(* IEC 61131-3 sources: POMIRTS_lab3/AS/Library/AsCisMan, 3 files *)

(* ---- AsCisMan.typ ---- *)
(********************************************************************
 * COPYRIGHT -- Bernecker + Rainer
 ********************************************************************
 * Library: AsCisMan
 * File: AsCisMan.typ
 * Author: B+R
 ********************************************************************
 * Data types of library AsCisMan
 ********************************************************************)

TYPE
	vfAxisInfo_typ : STRUCT								(*statistics and internal information*)
		Device	: STRING[20] ;							(*interface device string*)
		Mode	: STRING[20] ;							(*interface mode string*)
		Typ	: UINT ;									(*device type*)
		IndexVf	: USINT ;								(*internal array index for axis structure*)
		IndexIf	: USINT ;								(*internal array index for interface structure*)
		VersionLib	: ARRAY[0..9] OF USINT ;			(*version of the AsCisMan.br library*)
		VersionDrv	: ARRAY[0..9] OF USINT ;			(*version of the driver task cis_vf.br or cis_ps.br*)
		VersionOsVf	: ARRAY[0..9] OF USINT ;			(*version of the cis_osvf operating system transferred to the VF*)
		VersionData	: ARRAY[0..9] OF USINT ;			(*data object version*)
		VfPNominal	: UINT ;							(*nominal power of the VF module in W (read from the VF EPROM)*)
		VfModuleID	: UINT ;							(*ID number of the VF module (read from the VF EPROM)*)
		VfSerialNr	: UDINT ;							(*serial number of the VF module (read from the VF EPROM)*)
		VfCurrentLSB	: UINT ;						(*current resolution of VF module in mA/Bit (read from the VF EPROM)*)
		CyclesPowerOn	: UINT ;						(*counter for the number of power ons*)
		HoursPowerOn	: UDINT ;						(*counter for the hours that voltage is applied to the VF module*)
		HoursMotorOn	: UDINT ;						(*counter for the hours the motor has power*)
		MinutesPowerOn	: USINT ;						(*counter minutes of VF module under voltage (incremented to 254 only once)*)
		MinutesMotorOn	: USINT ;						(*counter minutes of powered motor (incremented to 254 only once)*)
		HistoryMaxTempIGBT	: USINT ;					(*overall maximum IGBT temperature in degree celsius*)
		HistoryMaxTempMotor	: USINT ;					(*overall maximum motor temperature in degree celsius*)
		HistoryMaxTempCPU1	: USINT ;					(*overall maximum CPU temperature1 in degree celsius*)
		HistoryMaxTempCPU2	: USINT ;					(*overall maximum CPU temperature2 in degree celsius*)
		HistoryMaxCurrent	: UINT ;					(*overall maximum DC bus current in mA*)
		HistoryMaxUDCLink	: UINT ;					(*overall maximum DC bus voltage in VCD*)
		HistoryChangedSlot	: USINT ;					(*counter VF module inserted in different slot than at the last power on*)
		HistoryChangedPS	: USINT ;					(*counter VF module inserted in different CIS PS than at the last power on*)
		FactUDCLink	: REAL ;							(*DC bus voltage measurement correction factor (0.880-1.120)*)
		IdentXOpen	: UDINT ;							(*internal use*)
		StatusXOpen	: UINT ;							(*internal use*)
		IdentData	: UDINT ;							(*internal use*)
		pData	: UDINT ;								(*internal use*)
		lenData	: UDINT ;								(*internal use*)
		StatusData	: UINT ;							(*internal use*)
	END_STRUCT;
	vfAxisNetwork_typ : STRUCT							(*network and individual parameter operations*)
		Init	: USINT ;								(*initializes the connection (FU responds to the driver)*)
		ParIDRequest	: USINT ;						(*sets/reads FI parameters: requested ID*)
		ParIDResponse	: USINT ;						(*sets/reads individual parameters: response from read/write ID*)
		ParData	: UINT ;								(*sets/reads individual parameters depending on the parameter: data*)
		EPromAdrRequest	: USINT ;						(*sets/reads byte at EEPROM: requested address ($00…$7F reserved for OS)*)
		EPromAdrResponse	: USINT ;					(*sets/reads EEPROM bytes: response from read/write address*)
		EPromData	: USINT ;							(*sets/reads EEPROM : Data*)
	END_STRUCT;
	vfAxisParaVf_typ : STRUCT							(*parameter*)
		UDCNominal	: UINT ;							(*nominal DC bus voltage*)
		VfCurveV	: ARRAY[0..7] OF UINT ;				(*v/f curve array (voltage point 0-7)*)
		VfCurveF	: ARRAY[0..7] OF UINT ;				(*v/f curve array (frequency point 0-7)*)
		FreqMax	: UINT ;								(*maximum frequency*)
		MaxCurrent	: UINT ;							(*DC bus current limit*)
		IntAccRamp	: UINT ;							(*internal acceleration ramp (corresponds to about 5 ms/step)*)
		IntDecRamp	: UINT ;							(*internal deceleration ramp (corresponds to about 5 ms/step)*)
		TimeStopped	: UINT ;							(*time between the motor's stopping and status, stopped = 1*)
		ModeStopped	: USINT ;							(*ModeStopped=0..speed takes effect immediately, ModeStopped=1..speed takes effect only when status*)
		Pwm	: USINT ;									(*frequency for pulse width modulation (currently fixed at 5 kHz)*)
		TorqueCtrl	: USINT ;							(*enable VF torque check*)
		TempMotorMax	: USINT ;						(*maximum motor temperature*)
		CurErrorAutoAck	: USINT ;						(*enables automatic acknowledgement of overcurrent errors*)
		spare1	: USINT ;								(*free*)
		UDCMax	: UINT ;								(*maximum permissible DC bus voltage: 0...default value 760VDC is used*)
	END_STRUCT;
	vfAxisParaTemp_typ : STRUCT							(*parameter*)
		R0	: UINT ;									(*resistance for T[0]*)
		R7	: UINT ;									(*resistance for T[7]*)
		T	: ARRAY[0..7] OF SINT ;						(*field for temperature*)
	END_STRUCT;
	vfAxisPara_typ : STRUCT								(*parameter*)
		Vf	: vfAxisParaVf_typ ;						(*CIS FU parameters*)
		Temp	: vfAxisParaTemp_typ ;					(*motor temperature sensor parameter*)
	END_STRUCT;
	vfAxisMove_typ : STRUCT								(*motion*)
		Speed	: DINT ;								(*target speed [0.01Hz] (-600.00…600.00Hz)*)
		CurrLimit	: UINT ;							(*DC bus current limit (0…65000mA)*)
		UDCInject	: UINT ;							(*DC brake voltage (for StopMode=2 only)*)
		StopMode	: USINT ;							(*is given es a target speed, e.g. 0...motor loses current immediately and spins out*)
		AccPos	: UDINT ;								(*acceleration in a positive direction [0.01Hz/s] (0.01…1000.00Hz/s)*)
		AccNeg	: UDINT ;								(*acceleration in a negative direction [0.01Hz/s] (0.01…1000.00Hz/s)*)
		DecPos	: UDINT ;								(*deceleration in a positive direction [0.01Hz/s] (0.01…1000.00Hz/s)*)
		DecNeg	: UDINT ;								(*deceleration in a negative direction [0.01Hz/s] (0.01…1000.00Hz/s)*)
	END_STRUCT;
	vfAxisStatus_typ : STRUCT							(*status*)
		SpeedRamped	: DINT ;							(*current ramp speed being sent to the FC (unit = 0.01Hz)*)
		UDCInject	: UINT ;							(*currently induced braking voltage in V*)
		ActTempIGBT	: USINT ;							(*current FC-IGBT temperature in degree celsius*)
		MaxTempIGBT	: USINT ;							(*maximum FC-IGBT temperature in degree celsius*)
		ActTempMotor	: USINT ;						(*current FC motor temperature in degree celsius*)
		MaxTempMotor	: USINT ;						(*maximum FC motor temperature in degree celsius*)
		ActTempRect	: USINT ;							(*current bridge rectifier temperature in degree celsius*)
		MaxTempRect	: USINT ;							(*maximum bridge rectifier temperature in degree celsius*)
		ActTempPS	: USINT ;							(*current internal temperature in degree celsius*)
		MaxTempPS	: USINT ;							(*maximum internal temperature in degree celsius*)
		ActTempCPU1	: USINT ;							(*current internal CIS CPU temperature 1 in degree celsius (up to 80degree OK)*)
		MaxTempCPU1	: USINT ;							(*maximum internal CIS CPU temperature 1 in degree celsius*)
		ActTempCPU2	: USINT ;							(*current internal CIS CPU temperature 2 in degree celsius (up to 80degree OK)*)
		MaxTempCPU2	: USINT ;							(*maximum internal CIS CPU temperature 2 in degree celsius*)
		ActCurrent	: UINT ;							(*current IGBT DC bus current in mA*)
		MaxCurrent	: UINT ;							(*maximum IGBT DC bus current in mA*)
		ActUDCLink	: UINT ;							(*current FC DC bus voltage in VDC*)
		MaxUDCLink	: UINT ;							(*maximum FC DC bus voltage in VDC*)
		CPU	: UINT ;									(*statusBits CPU*)
		CISPS1	: USINT ;								(*statusBits1 FC basis board*)
		CISPS2	: USINT ;								(*statusBits2 FC basis board*)
		Stopped	: USINT ;								(*Motor stopped (current rotor speed = 0 detected)*)
		Active	: USINT ;								(*FC active (cyclic speed assignment to CIS FC is active)*)
		ParaInit	: USINT ;							(*Parameter initialized*)
		PowerOk	: USINT ;								(*DC bus voltage OK*)
	END_STRUCT;
	vfAxisError_typ : STRUCT							(*error*)
		Active	: USINT ;								(*cumulative error: at least one error is active*)
		Current	: USINT ;								(*DC bus current over current limit (warning)*)
		CurrentOff	: USINT ;							(*DC bus current too high - FC stopped, error must be acknowledged*)
		TempIGBT	: USINT ;							(*IGBT temperature warning*)
		TempIGBTOff	: USINT ;							(*IGBT temperature too high - FC stopped, error must be acknowledged*)
		TempMotor	: USINT ;							(*motor temperature warning*)
		TempMotorOff	: USINT ;						(*motor temperature too high - FC stopped, error must be acknowledged*)
		TempMotorBreak	: USINT ;						(*motor temperature sensor wire break*)
		TempMotorShort	: USINT ;						(*motor temperature sensor short circuit*)
		VoltageHigh	: USINT ;							(*DC bus voltage too high*)
		Amplifier	: USINT ;							(*IGBT control internal error*)
		cntComTimeOff	: UDINT ;						(*counter: milliseconds that have passed since the last valid response from the FC*)
		cntCom	: UINT ;								(*counter communication error: communication timeout*)
		cntCommand	: UINT ;							(*counter communication error: illegal command*)
		cntParameter	: UINT ;						(*counter communication error: parameter outside of the permitted range*)
		cntService	: UINT ;							(*counter communication error: illegal service command*)
		cntAcknowledge	: UINT ;						(*counter communication error: could not acknowledge error - error still active*)
		cntCheckSumVFD	: UINT ;						(*counter checksum error (illegal checksum in FC data)*)
		cntEpromLock	: UINT ;						(*counter communication error: EPROM access blocked*)
		cntAmplitudeDelta	: UINT ;					(*counter error in VF curve parameters (voltage amplitude not climbing monotonously)*)
		cntFrequencyDelta	: UINT ;					(*counter error in VF curve parameters (frequency not climbing monotonously)*)
		cntLifeSignal	: UINT ;						(*counter: FC didn't receive any valid data for 200 ms*)
		cntCheckSumCPU	: UINT ;						(*counter checksum error (illegal checksum in FC data)*)
		cntResponsePara	: UINT ;						(*counter communication error (illegal data in response telegram)*)
		cntResponseSpd	: UINT ;						(*counter communication error (illegal data in response telegram)*)
		cntResponseError	: UINT ;					(*counter communication error (illegal data in response telegram)*)
	END_STRUCT;
	vfAxisInterntOut_typ : STRUCT						(*internal use*)
		IN	: BOOL ;
		PT	: UDINT ;
		Q	: BOOL ;
		ET	: UDINT ;
		StartTime	: UDINT ;
		M	: BOOL ;
	END_STRUCT;
	vfAxisInternal_typ : STRUCT							(*internal use*)
		cmdSubject	: UINT ;							(*handshake for the vfaction() function: command subject*)
		cmdAction	: UINT ;							(*handshake for the vfaction() function: command action*)
		cmdPara	: USINT ;								(*handshake for the vfaction() function: command related parameterID*)
		cmdData	: UINT ;								(*handshake for the vfaction() function: command related data*)
		cntStep	: USINT ;								(*internal step*)
		Write	: USINT ;								(*0..process command, 1..send frame, 2..wait for response*)
		BufWrite	: ARRAY[0..5] OF USINT ;			(*buffer for the sent frame*)
		BufRead	: ARRAY[0..5] OF USINT ;				(*buffer for the received frame*)
		Sequence	: USINT ;							(*indicates the class of parameter ID*)
		cntInitEpromRead	: USINT ;					(*counter for read EPROM data during initialization*)
		cntInitUfCurveSet	: USINT ;					(*counter for sent U/f data*)
		tOut	: vfAxisInterntOut_typ ;				(*receive timeout*)
		ActTempMotorR	: UINT ;						(*measured resistance of the motor temperature sensor*)
		MaxTempMotorR	: UINT ;						(*measured resistance of the motor temperature sensor*)
		TempMotorRFilter	: ARRAY[0..9] OF UINT ;		(*filter buffer for motor temperature filters*)
		cntTempMotorRFilter	: UINT ;					(*filter counter for motor temperature filters*)
		OldUDCInject	: UINT ;						(*UDCInject edge*)
		SpeedRamped	: REAL ;							(*output of the speed ramp in REAL*)
		TestFan	: USINT ;								(*=1 for manually testing the internal fans*)
		cntInfoWrite	: USINT ;						(*counter*)
		CyclesPowerOnCheck	: UINT ;					(*EPROM: backup copy of Info.CyclesPowerOn*)
		HoursPowerOnCheck	: UDINT ;					(*EPROM: backup copy of Info.HoursPowerOn*)
		HoursMotorOnCheck	: UDINT ;					(*EPROM: backup copy of Info.HoursMotorOn*)
		HistoryBufferAdr	: ARRAY[0..15] OF USINT ;	(*history address storage*)
		HistoryBufferData	: ARRAY[0..15] OF USINT ;	(*history data storage*)
		HistoryBufferCnt	: USINT ;					(*counter for pending historical data*)
		HistorySlot	: USINT ;							(*EPROM: VF inserted in slot number*)
		HistoryMacId	: ARRAY[0..2] OF USINT ;		(*EPROM: MacID of the CIS-PS*)
		HistoryMacIdChecksum	: USINT ;				(*EPROM: MacID checksum*)
		FactUDCLink	: REAL ;							(*EPROM: DC bus voltage measurement correction factor*)
	END_STRUCT;
	vfAXIS_typ : STRUCT									(*AXIS information*)
		Info	: vfAxisInfo_typ ;						(*statistics and internal information*)
		Network	: vfAxisNetwork_typ ;					(*network and individual parameter operations*)
		Para	: vfAxisPara_typ ;						(*parameter*)
		Move	: vfAxisMove_typ ;						(*motion*)
		Status	: vfAxisStatus_typ ;					(*status*)
		Error	: vfAxisError_typ ;						(*error*)
		Internal	: vfAxisInternal_typ ;				(*internal use*)
	END_STRUCT;
	vfInterfaceBuf_typ : STRUCT							(*internal use*)
		Byte0	: USINT ;
		Command	: USINT ;
		ByteHI	: USINT ;
		ByteLO	: USINT ;
		CheckSum	: USINT ;
		spare0	: USINT ;
	END_STRUCT;
	vfInterface_typ : STRUCT							(*internal use*)
		Ident	: UDINT ;
		cntFrame	: USINT ;
		oldFrame	: USINT ;
		cntBufWrite	: USINT ;
		cntBufRead	: USINT ;
		cntFrameWrite	: USINT ;
		cntFrameRead	: USINT ;
		FrameRead	: ARRAY[0..7] OF USINT ;
		cntFrameRead85	: USINT ;
		FrameRead85	: ARRAY[0..1] OF USINT ;
		BufWrite	: ARRAY[0..7] OF vfInterfaceBuf_typ ;
		BufRead	: ARRAY[0..7] OF vfInterfaceBuf_typ ;
	END_STRUCT;
	vfDebug_typ : STRUCT								(*internal use*)
		Time	: UDINT ;
		UDC	: UINT ;
		Current	: UINT ;
		Temp	: USINT ;
		BufferSend	: ARRAY[0..4] OF USINT ;
		BufferRecv	: ARRAY[0..11] OF USINT ;
		BufferRecvNb	: USINT ;
		ErrorCom	: USINT ;
		ErrorCheckFU	: USINT ;
		ErrorCheckCPU	: USINT ;
		ErrorCommand	: USINT ;
		ErrorParameter	: USINT ;
		ErrorService	: USINT ;
		ErrorResponse	: USINT ;
		ErrorAcknowledge	: USINT ;
		ErrorEpromLock	: USINT ;
		ErrorAmplitudeDelta	: USINT ;
		ErrorFrequencyDelta	: USINT ;
		ErrorLifeSignal	: USINT ;
	END_STRUCT;
	vfDebugResponse_typ : STRUCT						(*internal use*)
		Write	: ARRAY[0..5] OF USINT ;
		Read	: ARRAY[0..5] OF USINT ;
	END_STRUCT;
	vfErrorTrace_typ : STRUCT							(*internal use*)
		Fu	: USINT ;
		Error	: USINT ;
		Time	: UDINT ;
	END_STRUCT;
END_TYPE

(* ---- AsCisMan.fun ---- *)
(********************************************************************
 * COPYRIGHT -- Bernecker + Rainer
 ********************************************************************
 * Library: AsCisMan
 * File: AsCisMan.fun
 * Author: B+R
 ********************************************************************
 * Functions and function blocks of library AsCisMan
 ********************************************************************)

FUNCTION_BLOCK initps05								(*boots and allocates a CIS base unit 80CIS.PS0-5 (7 slot, 6.5 kW)*)
	VAR_INPUT
		Enable	:BOOL;								(*enables execution*)
		ParaVF1	:STRING[8];							(*name of the slot1 initialization parameter data object*)
		ParaVF2	:STRING[8];							(*name of the slot2 initialization parameter data object*)
		ParaVF3	:STRING[8];							(*name of the slot3 initialization parameter data object*)
		ParaVF4	:STRING[8];							(*name of the slot4 initialization parameter data object*)
		ParaVF5	:STRING[8];							(*name of the slot5 initialization parameter data object*)
		ParaVF6	:STRING[8];							(*name of the slot6 initialization parameter data object*)
		ParaVF7	:STRING[8];							(*name of the slot7 initialization parameter data object*)
	END_VAR
	VAR_OUTPUT
		Status	:UINT;								(*execution status: ERR_OK, ERR_FUB_ENABLE_FALSE, 0xXXXX = see help*)
		IdentCPU	:UDINT;							(*identifier for the CPU data (for use with run_cpu)*)
		IdentVF1	:UDINT;							(*identifier for the VF slot 1 (for use with run_vfx)*)
		IdentVF2	:UDINT;							(*identifier for the VF slot 2 (for use with run_vfx)*)
		IdentVF3	:UDINT;							(*identifier for the VF slot 3 (for use with run_vfx)*)
		IdentVF4	:UDINT;							(*identifier for the VF slot 4 (for use with run_vfx)*)
		IdentVF5	:UDINT;							(*identifier for the VF slot 5 (for use with run_vfx)*)
		IdentVF6	:UDINT;							(*identifier for the VF slot 6 (for use with run_vfx)*)
		IdentVF7	:UDINT;							(*identifier for the VF slot 7 (for use with run_vfx)*)
		BootOkBitsVF	:USINT;						(*bit-coded status: bit=0...boot failed, bit=1...boot successful*)
	END_VAR
	VAR
		Object	:ARRAY[0..8] OF UDINT;				(*internal variable*)
		StatusAlloc	:ARRAY[0..8] OF UINT;			(*internal variable*)
			vf_bsl_00	:vf_bsl;					(*internal variable*)
			vf_bsl_01	:vf_bsl;					(*internal variable*)
		vf_bsl_02	:vf_bsl;						(*internal variable*)
		vf_bsl_03	:vf_bsl;						(*internal variable*)
		vf_bsl_04	:vf_bsl;						(*internal variable*)
		vf_bsl_05	:vf_bsl;						(*internal variable*)
		vf_bsl_06	:vf_bsl;						(*internal variable*)
		vf_bsl_07	:vf_bsl;						(*internal variable*)
		vf_bsl_08	:vf_bsl;						(*internal variable*)
		zzvfalloc00000	:vfalloc;					(*internal variable*)
		zzvfalloc00001	:vfalloc;					(*internal variable*)
		zzvfalloc00002	:vfalloc;					(*internal variable*)
		zzvfalloc00003	:vfalloc;					(*internal variable*)
		zzvfalloc00004	:vfalloc;					(*internal variable*)
		zzvfalloc00005	:vfalloc;					(*internal variable*)
		zzvfalloc00006	:vfalloc;					(*internal variable*)
		zzvfalloc00007	:vfalloc;					(*internal variable*)
	END_VAR
END_FUNCTION_BLOCK

FUNCTION_BLOCK initps04								(*boots and allocates a CIS base unit 80CIS.PS0-4 (4 slot, 16 kW)*)
	VAR_INPUT
		Enable	:BOOL;								(*enables execution*)
		ParaVF1	:STRING[8];							(*name of the slot1 initialization parameter data object*)
		ParaVF2	:STRING[8];							(*name of the slot2 initialization parameter data object*)
		ParaVF3	:STRING[8];							(*name of the slot3 initialization parameter data object*)
		ParaVF4	:STRING[8];							(*name of the slot4 initialization parameter data object*)
	END_VAR
	VAR_OUTPUT
		Status	:UINT;								(*execution status: ERR_OK, ERR_FUB_ENABLE_FALSE, 0xXXXX = see help*)
		IdentCPU	:UDINT;							(*identifier for the CPU data (for use with run_cpu)*)
		IdentVF1	:UDINT;							(*identifier for the VF slot 1 (for use with run_vfx)*)
		IdentVF2	:UDINT;							(*identifier for the VF slot 2 (for use with run_vfx)*)
		IdentVF3	:UDINT;							(*identifier for the VF slot 3 (for use with run_vfx)*)
		IdentVF4	:UDINT;							(*identifier for the VF slot 4 (for use with run_vfx)*)
		BootOkBitsVF	:USINT;						(*bit-coded status: bit=0...boot failed, bit=1...boot successful*)
	END_VAR
	VAR
		Object	:ARRAY[0..8] OF UDINT;				(*internal variable*)
		StatusAlloc	:ARRAY[0..8] OF UINT;			(*internal variable*)
		vf_bsl_00	:vf_bsl;						(*internal variable*)
		vf_bsl_01	:vf_bsl;						(*internal variable*)
		vf_bsl_02	:vf_bsl;						(*internal variable*)
		vf_bsl_03	:vf_bsl;						(*internal variable*)
		vf_bsl_08	:vf_bsl;						(*internal variable*)
		zzvfalloc00000	:vfalloc;					(*internal variable*)
		zzvfalloc00001	:vfalloc;					(*internal variable*)
		zzvfalloc00002	:vfalloc;					(*internal variable*)
		zzvfalloc00003	:vfalloc;					(*internal variable*)
		zzvfalloc00004	:vfalloc;					(*internal variable*)
	END_VAR
END_FUNCTION_BLOCK

FUNCTION_BLOCK initps03								(*boots and allocates a CIS base unit 80CIS.PS0-3 (8 slot, 16 kW)*)
	VAR_INPUT
		Enable	:BOOL;								(*enables execution*)
		ParaVF1	:STRING[8];							(*name of the slot1 initialization parameter data object*)
		ParaVF2	:STRING[8];							(*name of the slot2 initialization parameter data object*)
		ParaVF3	:STRING[8];							(*name of the slot3 initialization parameter data object*)
		ParaVF4	:STRING[8];							(*name of the slot4 initialization parameter data object*)
		ParaVF5	:STRING[8];							(*name of the slot5 initialization parameter data object*)
		ParaVF6	:STRING[8];							(*name of the slot6 initialization parameter data object*)
		ParaVF7	:STRING[8];							(*name of the slot7 initialization parameter data object*)
		ParaVF8	:STRING[8];							(*name of the slot8 initialization parameter data object*)
	END_VAR
	VAR_OUTPUT
		Status	:UINT;								(*execution status: ERR_OK, ERR_FUB_ENABLE_FALSE, 0xXXXX = see help*)
		IdentCPU	:UDINT;							(*identifier for the CPU data (for use with run_cpu)*)
		IdentVF1	:UDINT;							(*identifier for the VF slot 1 (for use with run_vfx)*)
		IdentVF2	:UDINT;							(*identifier for the VF slot 2 (for use with run_vfx)*)
		IdentVF3	:UDINT;							(*identifier for the VF slot 3 (for use with run_vfx)*)
		IdentVF4	:UDINT;							(*identifier for the VF slot 4 (for use with run_vfx)*)
		IdentVF5	:UDINT;							(*identifier for the VF slot 5 (for use with run_vfx)*)
		IdentVF6	:UDINT;							(*identifier for the VF slot 6 (for use with run_vfx)*)
		IdentVF7	:UDINT;							(*identifier for the VF slot 7 (for use with run_vfx)*)
		IdentVF8	:UDINT;							(*identifier for the VF slot 8 (for use with run_vfx)*)
		BootOkBitsVF	:USINT;						(*bit-coded status: bit=0...boot failed, bit=1...boot successful*)
	END_VAR
	VAR
		Object	:ARRAY[0..8] OF UDINT;				(*internal variable*)
		StatusAlloc	:ARRAY[0..8] OF UINT;			(*internal variable*)
		vf_bsl_00	:vf_bsl;						(*internal variable*)
		vf_bsl_01	:vf_bsl;						(*internal variable*)
		vf_bsl_02	:vf_bsl;						(*internal variable*)
		vf_bsl_03	:vf_bsl;						(*internal variable*)
		vf_bsl_04	:vf_bsl;						(*internal variable*)
		vf_bsl_05	:vf_bsl;						(*internal variable*)
		vf_bsl_06	:vf_bsl;						(*internal variable*)
		vf_bsl_07	:vf_bsl;						(*internal variable*)
		vf_bsl_08	:vf_bsl;						(*internal variable*)
		zzvfalloc00000	:vfalloc;					(*internal variable*)
		zzvfalloc00001	:vfalloc;					(*internal variable*)
		zzvfalloc00002	:vfalloc;					(*internal variable*)
		zzvfalloc00003	:vfalloc;					(*internal variable*)
		zzvfalloc00004	:vfalloc;					(*internal variable*)
		zzvfalloc00005	:vfalloc;					(*internal variable*)
		zzvfalloc00006	:vfalloc;					(*internal variable*)
		zzvfalloc00007	:vfalloc;					(*internal variable*)
		zzvfalloc00008	:vfalloc;					(*internal variable*)
	END_VAR
END_FUNCTION_BLOCK

FUNCTION_BLOCK initps02								(*boots and allocates a CIS base unit 80CIS.PS0-2 (8 slot, 8 kW)*)
	VAR_INPUT
		Enable	:BOOL;								(*enables execution*)
		ParaVF1	:STRING[8];							(*name of the slot1 initialization parameter data object*)
		ParaVF2	:STRING[8];							(*name of the slot2 initialization parameter data object*)
		ParaVF3	:STRING[8];							(*name of the slot3 initialization parameter data object*)
		ParaVF4	:STRING[8];							(*name of the slot4 initialization parameter data object*)
		ParaVF5	:STRING[8];							(*name of the slot5 initialization parameter data object*)
		ParaVF6	:STRING[8];							(*name of the slot6 initialization parameter data object*)
		ParaVF7	:STRING[8];							(*name of the slot7 initialization parameter data object*)
		ParaVF8	:STRING[8];							(*name of the slot8 initialization parameter data object*)
	END_VAR
	VAR_OUTPUT
		Status	:UINT;								(*execution status: ERR_OK, ERR_FUB_ENABLE_FALSE, 0xXXXX = see help*)
		IdentCPU	:UDINT;							(*identifier for the CPU data (for use with run_cpu)*)
		IdentVF1	:UDINT;							(*identifier for the VF slot 1 (for use with run_vfx)*)
		IdentVF2	:UDINT;							(*identifier for the VF slot 2 (for use with run_vfx)*)
		IdentVF3	:UDINT;							(*identifier for the VF slot 3 (for use with run_vfx)*)
		IdentVF4	:UDINT;							(*identifier for the VF slot 4 (for use with run_vfx)*)
		IdentVF5	:UDINT;							(*identifier for the VF slot 5 (for use with run_vfx)*)
		IdentVF6	:UDINT;							(*identifier for the VF slot 6 (for use with run_vfx)*)
		IdentVF7	:UDINT;							(*identifier for the VF slot 7 (for use with run_vfx)*)
		IdentVF8	:UDINT;							(*identifier for the VF slot 8 (for use with run_vfx)*)
		BootOkBitsVF	:USINT;						(*bit-coded status: bit=0...boot failed, bit=1...boot successful*)
	END_VAR
	VAR
		Object	:ARRAY[0..8] OF UDINT;				(*internal variable*)
		StatusAlloc	:ARRAY[0..8] OF UINT;			(*internal variable*)
		vf_bsl_00	:vf_bsl;						(*internal variable*)
		vf_bsl_01	:vf_bsl;						(*internal variable*)
		vf_bsl_02	:vf_bsl;						(*internal variable*)
		vf_bsl_03	:vf_bsl;						(*internal variable*)
		vf_bsl_04	:vf_bsl;						(*internal variable*)
		vf_bsl_05	:vf_bsl;						(*internal variable*)
		vf_bsl_06	:vf_bsl;						(*internal variable*)
		vf_bsl_07	:vf_bsl;						(*internal variable*)
		vf_bsl_08	:vf_bsl;						(*internal variable*)
		zzvfalloc00000	:vfalloc;					(*internal variable*)
		zzvfalloc00001	:vfalloc;					(*internal variable*)
		zzvfalloc00002	:vfalloc;					(*internal variable*)
		zzvfalloc00003	:vfalloc;					(*internal variable*)
		zzvfalloc00004	:vfalloc;					(*internal variable*)
		zzvfalloc00005	:vfalloc;					(*internal variable*)
		zzvfalloc00006	:vfalloc;					(*internal variable*)
		zzvfalloc00007	:vfalloc;					(*internal variable*)
		zzvfalloc00008	:vfalloc;					(*internal variable*)
	END_VAR
END_FUNCTION_BLOCK

FUNCTION_BLOCK run_cpu								(*communicates cyclic to the CPU*)
	VAR_INPUT
		Enable	:BOOL;								(*enables execution*)
		IdentCPU	:UDINT;							(*identifier for the CPU data (from initps0x)*)
	END_VAR
	VAR_OUTPUT
		Status	:UINT;								(*execution status: ERR_OK, ERR_FUB_ENABLE_FALSE, 0xXXXX = see help*)
		StatusBitsCPU	:UINT;						(*CPU register: bit 1: 0...24VDC OK, bit 1: 1...24V ERROR, bit 10: 1...DC*)
		ActUDCLink	:UINT;							(*current DC bus voltage measured in the CIS-PS*)
		ActTempCPU1	:USINT;							(*current CPU temperature 1*)
		ActTempCPU2	:USINT;							(*current CPU temperature 2*)
		ActTempRect	:USINT;							(*current bridge rectifier temperature*)
	END_VAR
	VAR
		dAxis	:REFERENCE TO vfAXIS_typ;			(*internal variable*)
	END_VAR
END_FUNCTION_BLOCK

FUNCTION_BLOCK run_vfx								(*communicates cyclic to an individual FI*)
	VAR_INPUT
		Enable	:BOOL;								(*enables execution*)
		IdentVF	:UDINT;								(*identifier for the VF data (from initps0x)*)
		AccPos	:REAL;								(*acceleration in positive direction*)
		DecPos	:REAL;								(*deceleration in positive direction*)
		AccNeg	:REAL;								(*acceleration in negative direction*)
		DecNeg	:REAL;								(*deceleration in negative direction*)
		SetSpeed	:REAL;							(*target speed*)
		SetCurrent	:UINT;							(*DC bus current limit*)
		SetUDCInject	:UINT;						(*DC brake voltage (for StopMode=2 only)*)
		StopMode	:USINT;							(*e.g. StopMode=0...motor loses current immediately and spins out*)
		CmdErrorAck	:BOOL;							(*acknowledge error command (level-sensitive)*)
	END_VAR
	VAR_OUTPUT
		Status	:UINT;								(*execution status: ERR_OK, ERR_FUB_ENABLE_FALSE, 0xXXXX = see help*)
		ActSpeed	:REAL;							(*current ramp speed being sent to the FC*)
		ActCurrent	:UINT;							(*current IGBT DC bus current*)
		ActUDCInject	:UINT;						(*currently provided braking voltage*)
		ActTempIGBT	:USINT;							(*current FC-IGBT temperature*)
		ActTempMotor	:USINT;						(*current FC motor temperature*)
		ActUDCLink	:UINT;							(*current DC bus voltage measured in the VF*)
		Stopped	:BOOL;								(*motor stopped (current rotor speed = 0 detected)*)
		ParaInit	:BOOL;							(*parameter initialized*)
		ErrorActive	:BOOL;							(*cumulative error: at least one error is active*)
		ErrorCurrent	:BOOL;						(*DC bus current over current limit (warning)*)
		ErrorCurrentOff	:BOOL;						(*DC bus current too high*)
		ErrorTempIGBT	:BOOL;						(*IGBT temperature warning*)
		ErrorTempIGBTOff	:BOOL;					(*IGBT temperature too high*)
		ErrorTempMotor	:BOOL;						(*motor temperature warning*)
		ErrorTempMotorOff	:BOOL;					(*motor temperature too high*)
		ErrorTempMotorBreak	:BOOL;					(*motor temperature sensor wire break*)
		ErrorTempMotorShort	:BOOL;					(*motor temperature sensor short circuit*)
		ErrorVoltageHigh	:BOOL;					(*DC bus voltage too high*)
		ErrorAmplifier	:BOOL;						(*IGBT control internal error*)
		ErrorCntComTimeOff	:UDINT;					(*counter: milliseconds that have passed since the last valid response from the FC*)
	END_VAR
	VAR
		step	:USINT;								(*internal variable*)
		StatusAction	:UINT;						(*internal variable*)
		dAxis	:REFERENCE TO vfAXIS_typ;			(*internal variable*)
	END_VAR
END_FUNCTION_BLOCK

FUNCTION vfinternal : UINT							(*internal use*)
	VAR_INPUT
		Data	:UDINT;								(*internal variable*)
	END_VAR
	VAR
		FubExtern	:REFERENCE TO ARRAY[0..19] OF UDINT;	(*internal variable*)
		SINT1	:SINT;								(*internal variable*)
		SINT2	:SINT;								(*internal variable*)
		UINT1	:UINT;								(*internal variable*)
		UINT2	:UINT;								(*internal variable*)
		UDINT1	:UDINT;								(*internal variable*)
		UDINT2	:UDINT;								(*internal variable*)
		zzRTInfo00000	:RTInfo;					(*internal variable*)
		UDINT_ETH1: UDINT;    						(*internal variable*)
		UDINT_ETH2: UDINT;    						(*internal variable*)
		UDINT_ETH3: UDINT;    						(*internal variable*)
	END_VAR
END_FUNCTION

FUNCTION_BLOCK vfalloc								(*allocates the FI object - used in initps02(), initps03(), initps04() and initps05()*)
	VAR_INPUT
		Interface	:UINT;							(*PLC bus ID*)
		Device	:UDINT;								(*device name given as a pointer*)
		Mode	:UDINT;								(*mode string given as a pointer*)
		Data	:UDINT;								(*data object string given as a pointer*)
		Object	:REFERENCE TO UDINT;				(*pointer to the FI structure*)
	END_VAR
	VAR_OUTPUT
		vfalloc	:UINT;								(*error number*)
	END_VAR
	VAR
		i	:USINT;									(*internal variable*)
		dAxis	:REFERENCE TO vfAXIS_typ;			(*internal variable*)
		dAdrTableAxis	:REFERENCE TO UDINT;		(*internal variable*)
		pAdrTableAxis	:UDINT;						(*internal variable*)
		lenAdrTableAxis	:UDINT;						(*internal variable*)
		pAllocAxis	:UDINT;							(*internal variable*)
		dInterface	:REFERENCE TO vfInterface_typ;	(*internal variable*)
		dAdrTableIf	:REFERENCE TO UDINT;			(*internal variable*)
		pAdrTableIf	:UDINT;							(*internal variable*)
		lenAdrTableIf	:UDINT;						(*internal variable*)
		pAllocIf	:UDINT;							(*internal variable*)
		DatObjInfo_01	:DatObjInfo;				(*internal variable*)
		IndexIf	:USINT;								(*internal variable*)
		Ident	:UDINT;								(*internal variable*)
		DeviceString	:ARRAY[0..7] OF USINT;		(*internal variable*)
		MoVerStructLib	:MoVerStruc_typ;			(*internal variable*)
		MoVerStruct	:MoVerStruc_typ;				(*internal variable*)
		pBufferVersionOs	:UDINT;					(*internal variable*)
		lenBufferVersionOs	:UDINT;					(*internal variable*)
		dBufferVersionOs	: REFERENCE TO ARRAY[0..7] OF STRING[10];	(*internal variable*)
	END_VAR
END_FUNCTION_BLOCK

FUNCTION vfaction : UINT							(*calls an FI function (command to driver) - used in run_cpu() and run_vfx()*)
	VAR_INPUT
		Object	:UDINT;								(*FI object (from vfalloc())*)
		cmdSubject	:UINT;							(*subject to which the command is applied*)
		cmdAction	:UINT;							(*command to be executed*)
	END_VAR
	VAR
		dAxis	:REFERENCE TO vfAXIS_typ;			(*internal variable*)
	END_VAR
END_FUNCTION

FUNCTION_BLOCK vf_bsl								(*transfers operating system to the FIs - used in initps02(), initps03(), initps04() and initps05()*)
	VAR_INPUT
		Enable	:USINT;								(*enables execution*)
		Interface	:UINT;							(*PLC bus ID*)
		Device	:UDINT;								(*device name given as a pointer, e.g. "Uart0" for the FI in slot 1*)
		Mode	:UDINT;								(*pointer to the uart (fixed)*)
		Data	:UDINT;								(*pointer to the name of the operating system data object*)
	END_VAR
	VAR_OUTPUT
		TransferOk	:USINT;							(*bit-coded status: bit=0...boot failed, bit=1...boot successful*)
		Status	:UINT;								(*execution status: ERR_OK, ERR_FUB_ENABLE_FALSE, 0xXXXX = see help*)
	END_VAR
	VAR
		sTransfer	:UINT;							(*internal variable*)
		DatObjInfo_01	:DatObjInfo;				(*internal variable*)
		BufRead	:ARRAY[0..7] OF USINT;				(*internal variable*)
		BufWrite	:ARRAY[0..7] OF USINT;			(*internal variable*)
		DataHeader	:ARRAY[0..7] OF USINT;			(*internal variable*)
		DataOs	:ARRAY[0..99] OF USINT;				(*internal variable*)
		DataRead	:ARRAY[0..99] OF USINT;			(*internal variable*)
		DataTest	:USINT;							(*internal variable*)
		cntTimeOut	:UDINT;							(*internal variable*)
		pData	:UDINT;								(*internal variable*)
		dData	:REFERENCE TO ARRAY[0..99] OF USINT;	(*internal variable*)
		i	:USINT;									(*internal variable*)
		UartIdent	:USINT;							(*internal variable*)
		DeviceString	:ARRAY[0..7] OF USINT;		(*internal variable*)
		pUartData	:ARRAY[0..7] OF UDINT;			(*internal variable*)
		dUartData	:REFERENCE TO UINT;				(*internal variable*)
		dUartStatusSend	:REFERENCE TO ARRAY[0..1] OF USINT;	(*internal variable*)
		dUartStatusRead	:REFERENCE TO ARRAY[0..1] OF USINT;	(*internal variable*)
		cntFrameWrite	:UDINT;						(*internal variable*)
		cntFrameRead	:UDINT;						(*internal variable*)
		cntUartData	:UINT;							(*internal variable*)
		dUartFPGAControl	:REFERENCE TO UINT;		(*internal variable*)
		dUartSRAMData	:REFERENCE TO UINT;			(*internal variable*)
		dUartSRAMAddress	:REFERENCE TO UINT;		(*internal variable*)
		dUartBslControl	:REFERENCE TO UINT;			(*internal variable*)
		dUartBslStatus	:REFERENCE TO UINT;			(*internal variable*)
		UartBslStatus	:UINT;						(*internal variable*)
		UartData	:UINT;							(*internal variable*)
		StatusGetAdr	:UINT;						(*internal variable*)
		MoVerStruct	:MoVerStruc_typ;				(*internal variable*)
		pBufferVersionOs	:UDINT;					(*internal variable*)
		lenBufferVersionOs	:UDINT;					(*internal variable*)
		dBufferVersionOs	:REFERENCE TO ARRAY[0..7] OF STRING[10];	(*internal variable*)
		DelayStart	:UINT;							(*internal variable*)
		DelayEnd	:UINT;							(*internal variable*)
	END_VAR
END_FUNCTION_BLOCK

(* ---- AsCisMan.var ---- *)
(********************************************************************
 * COPYRIGHT -- Bernecker + Rainer
 ********************************************************************
 * Library: AsCisMan
 * File: AsCisMan.var
 * Author: B+R
 ********************************************************************
 * Local variables of library AsCisMan
 ********************************************************************)

VAR CONSTANT
	vfERR_MODULE_CISVF_NOTINSTALLED	: UINT	:= 31143;	(*error: "cis_vf" module not found*)
	vfERR_MODULE_CISPS_NOTINSTALLED	: UINT	:= 31144;	(*error: "cis_ps" module not found*)
	vfERR_VERSION_CISOSVF_INVALID	: UINT	:= 31161;	(*error: version of the "cis_osvf" module invalid*)
	vfERR_VERSION_CISOSPS_INVALID	: UINT	:= 31163;	(*error: version of the "cis_osps" module invalid*)
	vfERR_INSUFFICIENT_TMP_MEMORY	: UINT	:= 31146;	(*error: not enough temporary memory available*)
	vfERR_INITDATA_MODULENOTFOUND	: UINT	:= 31153;	(*error: init data object not found*)
	vfERR_VERSION_CISVF_INVALID	: UINT	:= 31160;		(*error: version of the "cis_vf" module invalid*)
	vfERR_VERSION_CISPS_INVALID	: UINT	:= 31162;		(*error: version of the "cis_ps" module invalid*)
	vfERR_OSDATA_MODULENOTFOUND	: UINT	:= 31159;		(*error: operating system data object not found*)
	vfERR_INITDATA_ILLPARAMETER	: UINT	:= 31152;		(*error: init data object not found*)
	vfERR_OSDATA_ILLPARAMETER	: UINT	:= 31158;		(*error: operating system data object not found*)
	vfERR_INITDATA_ILLOBJTYPE	: UINT	:= 31151;		(*error: init data object has wrong object type (not a data object)*)
	vfERR_INITDATA_ILLOBJECT	: UINT	:= 31150;		(*error: init data object not found*)
	vfERR_UART_OPENED_TWICE	: UINT	:= 31145;			(*error: FI slot already allocated*)
	vfERR_OSDATA_ILLOBJTYPE	: UINT	:= 31157;			(*error: operating system data object has wrong object type (not a data object)*)
	vfERR_INVALID_INTERFACE	: UINT	:= 31141;			(*error: invalid parameter interface*)
	vfERR_OSDATA_ILLOBJECT	: UINT	:= 31156;			(*error: operating system data object not found*)
	vfERR_INVALID_COMMAND	: UINT	:= 31142;			(*error: invalid command*)
	vfPAR_ACK_TEMP_MOTOR	: USINT	:= 20;				(*parameters: used internally*)
	vfERR_INVALID_OBJECT	: UINT	:= 31140;			(*error: invalid object*)
	vfPAR_CUR_ERROR_ACK	: USINT	:= 25;					(*parameters: acknowledge over-current errors*)
	vfPAR_ACK_TEMP_IGBT	: USINT	:= 19;					(*parameters: acknowledge IGBT temperature errors*)
	vfPAR_ACK_AMPLIFIER	: USINT	:= 18;					(*parameters: acknowledge output stage errors*)
	vfPAR_TIME_STOPPED	: USINT	:= 20;					(*parameters: timer standstill detection*)
	vfPAR_MODE_STOPPED	: USINT	:= 21;					(*parameters: speed applied only after standstill*)
	vfPAR_EPROM_UNLOCK	: USINT	:= 42;					(*parameters: deactivate EEProm lock*)
	vfERR_INITDATA_LEN	: UINT	:= 31154;				(*error: size of data object incorrect*)
	vfPAR_TORQUE_CTRL	: USINT	:= 30;					(*parameters: activate/deactivate towque controller*)
	vfPAR_READ_UDC600	: USINT	:= 4;					(*parameters: used internally*)
	vfPAR_READ_UDC350	: USINT	:= 3;					(*parameters: used internally*)
	vfPAR_READ_STATUS	: USINT	:= 5;					(*parameters: used internally*)
	vfPAR_EPROM_WRITE	: USINT	:= 41;					(*parameters: write EEProm data*)
	vfPAR_BOOST_VALUE	: USINT	:= 5;					(*parameters: used internally*)
	vfPAR_UFCURVE_U7	: USINT	:= 57;					(*parameters: U/f characteristic curve, coordinate 7, voltage*)
	vfPAR_UFCURVE_U6	: USINT	:= 56;					(*parameters: U/f characteristic curve, coordinate 6, voltage*)
	vfPAR_UFCURVE_U5	: USINT	:= 55;					(*parameters: U/f characteristic curve, coordinate 5, voltage*)
	vfPAR_UFCURVE_U4	: USINT	:= 54;					(*parameters: U/f characteristic curve, coordinate 4, voltage*)
	vfPAR_UFCURVE_U3	: USINT	:= 53;					(*parameters: U/f characteristic curve, coordinate 3, voltage*)
	vfPAR_UFCURVE_U2	: USINT	:= 52;					(*parameters: U/f characteristic curve, coordinate 2, voltage*)
	vfPAR_UFCURVE_U1	: USINT	:= 51;					(*parameters: U/f characteristic curve, coordinate 1, voltage*)
	vfPAR_UFCURVE_U0	: USINT	:= 50;					(*parameters: U/f characteristic curve, coordinate 0, voltage*)
	vfPAR_UFCURVE_F7	: USINT	:= 67;					(*parameters: U/f characteristic curve, coordinate 7, frequency*)
	vfPAR_UFCURVE_F6	: USINT	:= 66;					(*parameters: U/f characteristic curve, coordinate 6, frequency*)
	vfPAR_UFCURVE_F5	: USINT	:= 65;					(*parameters: U/f characteristic curve, coordinate 5, frequency*)
	vfPAR_UFCURVE_F4	: USINT	:= 64;					(*parameters: U/f characteristic curve, coordinate 4, frequency*)
	vfPAR_UFCURVE_F3	: USINT	:= 63;					(*parameters: U/f characteristic curve, coordinate 3, frequency*)
	vfPAR_UFCURVE_F2	: USINT	:= 62;					(*parameters: U/f characteristic curve, coordinate 2, frequency*)
	vfPAR_UFCURVE_F1	: USINT	:= 61;					(*parameters: U/f characteristic curve, coordinate 1, frequency*)
	vfPAR_UFCURVE_F0	: USINT	:= 60;					(*parameters: U/f characteristic curve, coordinate 0, frequency*)
	vfPAR_READ_TEMP2	: USINT	:= 2;					(*parameters: used internally*)
	vfPAR_READ_TEMP1	: USINT	:= 1;					(*parameters: used internally*)
	vfPAR_EPROM_READ	: USINT	:= 40;					(*parameters: read EEProm data*)
	vfPAR_DOWN_VALUE	: USINT	:= 10;					(*parameters: internal deceleration ramp*)
	vfPAR_BOOST_MODE	: USINT	:= 2;					(*parameters: used internally*)
	vfPAR_TEMP_MODE	: USINT	:= 6;						(*parameters: used internally*)
	vfPAR_SET_SPEED	: USINT	:= 200;						(*parameters: set value for frequency*)
	vfPAR_OSVERSION	: USINT	:= 201;						(*parameters: used internally*)
	vfPAR_MOD_CURVE	: USINT	:= 11;						(*parameters: used internally*)
	vfPAR_CUR_VALUE	: USINT	:= 7;						(*parameters: over-current limit*)
	vfPAR_ACK_OC_QS	: USINT	:= 18;						(*parameters: acknowledge errors*)
	vfERR_AXISTABLE	: UINT	:= 31147;					(*error: axis table error*)
	vfPAR_UP_VALUE	: USINT	:= 9;						(*parameters: internal acceleration ramp*)
	vfPAR_ACK_TEMP	: USINT	:= 19;						(*parameters: acknowledge temperature errors*)
	vfERR_INITDATA	: UINT	:= 31149;					(*error: init data object not found*)
	vfCURRENT_MOVE	: UINT	:= 135;						(*movement, without target position, with current limit*)
	vfPAR_AMP_LIM	: USINT	:= 8;						(*parameters: used internally*)
	vfERR_IFTABLE	: UINT	:= 31148;					(*error: interface table error*)
	vfACKNOWLEDGE	: UINT	:= 257;						(*acknowledge*)
	vfSPEED_MOVE	: UINT	:= 134;						(*relative positioning*)
	vfERR_OSDATA	: UINT	:= 31155;					(*error: operating system data object not found*)
	vfPAR_F_MAX	: USINT	:= 4;							(*parameters: used internally*)
	vfPAR_BRAKE	: USINT	:= 23;							(*parameters: activate brake*)
	vfTRANSFER	: UINT	:= 1;							(*transfer vf_bsl()*)
	vfREL_MOVE	: UINT	:= 131;							(*relative positioning*)
	vfPAR_F_RT	: USINT	:= 3;							(*parameters: used internally*)
	vfINTERNAL	: UINT	:= 4;							(*FI vf_bsl(), vfalloc()*)
	vfABS_MOVE	: UINT	:= 132;							(*move with absolute target position*)
	vfSERVICE	: UINT	:= 165;							(*service interface*)
	vfPAR_PWM	: USINT	:= 1;							(*parameters: used internally*)
	vfHOMING	: UINT	:= 106;							(*homing*)
	vfGLOBAL	: UINT	:= 4;							(*global*)
	vfACTIVE	: UINT	:= 65535;						(*active*)
	vfSTART	: UINT	:= 260;								(*start*)
	vfERROR	: UINT	:= 1;								(*error*)
	vfEPROM	: UINT	:= 2;								(*EEProm*)
	vfBASIS	: UINT	:= 10;								(*base module vf_bsl(), vfalloc()*)
	vfSTOP	: UINT	:= 261;								(*stop*)
	vfSAVE	: UINT	:= 341;								(*save*)
	vfREAD	: UINT	:= 265;								(*read*)
	vfMOVE	: UINT	:= 3;								(*motion*)
	vfLOAD	: UINT	:= 0;								(*load vf_bsl()*)
	vfINIT	: UINT	:= 512;								(*initialize*)
	vfDATA	: UINT	:= 1024;							(*data*)
	vfSET	: UINT	:= 264;								(*set*)
	vfOK	: UINT	:= 0;								(*OK*)
END_VAR
